// TwinCAT 3 PLC project NastroTrasportatore
// ProgramVersion: 3.1.4024.0
// libraries:
//   Tc2_Standard, * (Beckhoff Automation GmbH)
//   Tc2_System, * (Beckhoff Automation GmbH)
//   Tc3_Module, * (Beckhoff Automation GmbH)
// project tree:
//   DUTs/ STATI.TcDUT
//   GVLs/ IO.TcGVL
//   / PlcTask.TcTTO
//   POUs/ MAIN.TcPOU, MSF.TcPOU, Oscillatore.TcPOU
// real-time tasks:
//   TASK PlcTask: cycle T#10ms, priority 20, ADS port 350

CONFIGURATION NastroTrasportatore
    RESOURCE PLC ON TwinCAT3
        TASK PlcTask(INTERVAL := T#10ms, PRIORITY := 20);
        PROGRAM MAIN WITH PlcTask : MAIN;
    END_RESOURCE
END_CONFIGURATION

// ---- DUTs/STATI.TcDUT
{attribute 'qualified_only'}
{attribute 'strict'}

TYPE STATI :
(
	S0,
	S1,
	S2,
	S3,
	SE,
	SA
);
END_TYPE

// ---- GVLs/IO.TcGVL
{attribute 'qualified_only'}

VAR_GLOBAL
	start  : BOOL;
	stop   : BOOL;
	emg    : BOOL;
	ack    : BOOL;
	
	fc1    : BOOL;
	fc2    : BOOL;
	
	H1     : BOOL;
	HEMG   : BOOL;
	
	M      : BOOL;
	libero : BOOL;
END_VAR

// ---- POUs/MAIN.TcPOU
PROGRAM MAIN

VAR
END_VAR

END_PROGRAM

// ---- POUs/MSF.TcPOU
FUNCTION_BLOCK MSF

VAR_INPUT
	start  : BOOL;
	stop   : BOOL;
	emg    : BOOL;
	ack    : BOOL;
	fc1    : BOOL;
	fc2    : BOOL;
END_VAR

VAR_OUTPUT
	H1     : BOOL;
	HEMG   : BOOL;
	M      : BOOL;
	libero : BOOL;
END_VAR

VAR
	enable : BOOL;
	tr_S0_S1 : BOOL;
	tr_S1_S2 : BOOL;
	tr_S2_S3 : BOOL;
	tr_S3_S1 : BOOL;
	tr_S3_S0 : BOOL;
	tr_SE_SA : BOOL;
	tr_SA_S0 : BOOL;
	stato  : STATI := STATI.S0;
END_VAR

END_FUNCTION_BLOCK

// ---- POUs/Oscillatore.TcPOU
FUNCTION_BLOCK Oscillatore

VAR_INPUT
	enable : BOOL;
	t_high : TIME;
	t_low  : TIME;
END_VAR

VAR_OUTPUT
	q      : BOOL;
END_VAR

VAR
	t1     : TON();
	t2     : TON();
END_VAR

t1(in := enable, );

END_FUNCTION_BLOCK
